TYPE ST_3DMarkerPositionNoLabel :
STRUCT
	x : REAL;
	y : REAL;
	z : REAL;
	id : DINT;
END_STRUCT
END_TYPE

(* stored: Version 1.1.0.1, ProductVersion 3.1.4026.8
   DUT ST_3DMarkerPositionNoLabel: Id {dca5d82f-1abd-49e2-a997-33e191ce9ce0} *)
